// TIA Portal V17 export
// export: Created 2022-07-28T18:03:21.9990991Z, ExportSetting None, DisplayName Totally Integrated Automation Portal, DisplayVersion V17, DisplayName TIA Portal Openness, DisplayVersion V17, DisplayName TIA Portal Teamcenter Gateway, DisplayVersion V17, DisplayName TIA Portal Version Control Interface, DisplayVersion V17, DisplayName TIA Portal Test Suite Advanced, DisplayVersion V17, DisplayName SINAMICS Startdrive Advanced, DisplayVersion V17, DisplayName SINAMICS DCC, DisplayVersion V17, DisplayName SINAMICS Startdrive G130, G150, S120, S150, SINAMICS MV, S210, DisplayVersion V17, DisplayName SINAMICS Startdrive G110M, G120, G120C, G120D, G120P, G115D, DisplayVersion V17, DisplayName STEP 7 Professional, DisplayVersion V17, DisplayName SIMATIC Energy Suite, DisplayVersion V17, DisplayName STEP 7 CFC, DisplayVersion V17, DisplayName STEP 7 Safety, DisplayVersion V17, DisplayName WinCC Advanced / Unified PC, DisplayVersion V17, DisplayName SIMATIC Visualization Architect, DisplayVersion V17
TYPE "_SlideGate_Blow_StateHMI"
   STRUCT
      dw_STW { ExternalWritable := 'False'} : DWord;   // Status+Mode WORD
      dw_EEW { ExternalWritable := 'False'} : DWord;   // ExternalError WORD
      dw_ILW_Open { ExternalWritable := 'False'} : DWord;   // Interlock WORD Open
      dw_ILW_Close { ExternalWritable := 'False'} : DWord;   // Interlock WORD Close
      dw_CONFW { ExternalWritable := 'False'} : DWord;   // Bit config paremeterts
      dw_STW_1 { ExternalWritable := 'False'} : DWord;
      dw_STW_2 { ExternalWritable := 'False'} : DWord;
      w_ALW1 { ExternalWritable := 'False'} : Word;
      w_ALW2 { ExternalWritable := 'False'} : Word := 16#0000;
      w_ALW3 { ExternalWritable := 'False'} : Word := 16#0000;
      w_ALW4 { ExternalWritable := 'False'} : Word := 16#0000;
      w_ALW5 { ExternalWritable := 'False'} : Word := 16#0000;
   END_STRUCT;
END_TYPE
